TYPE Status_Kaeltemittel : (gasformig, flussig, uberhitzt, unterkuhlt);
END_TYPE

(* stored: Version 1.1.0.1, ProductVersion 3.1.4019.2
   DUT Status_Kaeltemittel: Id {c4b58e57-ebdb-452c-b17e-fba0cb6d2908} *)
